{attribute addProperty BoxType "EL3152--0000"}
{attribute addProperty Id "ChannelAT %I*ARRAY[0..1] OF Channel_A23A2BD94860WcStateAT %I*WcState_98A4DF7520.250InfoDataAT %I*InfoData_BC63D37F80100"}
{attribute addProperty CRC "2116811507"}
{attribute addProperty SizeInBites "130"}
{attribute addProperty SizeInBytes "16.25"}
TYPE EL3152_C619ACF8 :
STRUCT
	{attribute addProperty Name "Channel"}
	Channel : ARRAY[0..1] OF Channel_A23A2BD9;
	{attribute addProperty Name "WcState"}
	WcState : WcState_98A4DF75;
	{attribute addProperty Name "InfoData"}
	InfoData : InfoData_BC63D37F;
END_STRUCT
END_TYPE

(* stored: Version 1.2.0.0, ProductVersion 3.1.4024.9
   DUT EL3152_C619ACF8: Id {8511689f-7c72-4b22-9a4d-138e051d2bc0} *)
